SUBAPPLICATION Uebung_039 (* Subapplication Type *)
  (* Standard: 61499-2 *)
  (* Version 1.0, 2023-10-23, franz *)
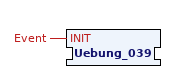
  EVENT_INPUT
    INIT;
  END_EVENT
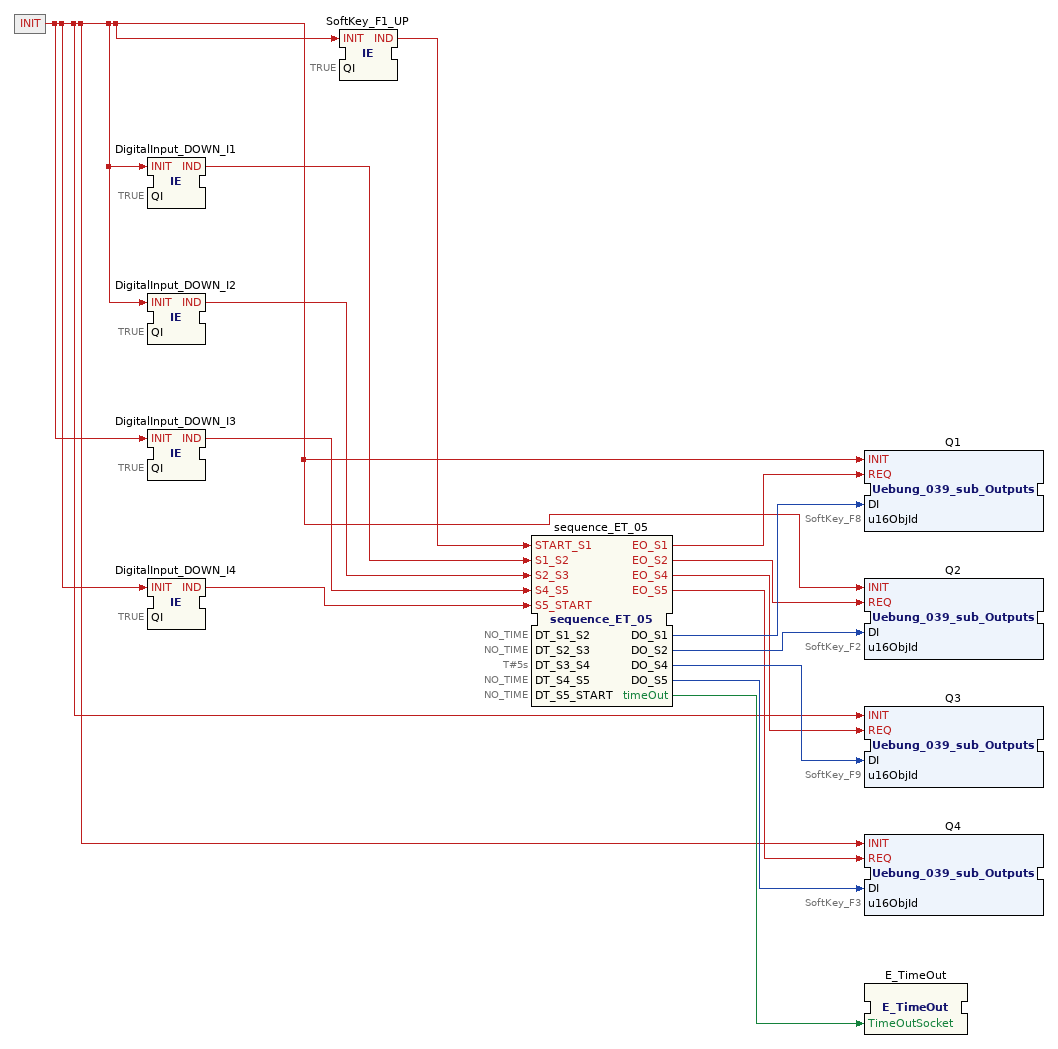
  FBS
    sequence_ET_05 : sequence_ET_05(DT_S1_S2 := NO_TIME, DT_S2_S3 := NO_TIME, DT_S3_S4 := T#5s, DT_S4_S5 := NO_TIME, DT_S5_START := NO_TIME);
    E_TimeOut : E_TimeOut;
    SoftKey_F1_UP : IE(QI := TRUE);
    DigitalInput_DOWN_I1 : IE(QI := TRUE);
    DigitalInput_DOWN_I2 : IE(QI := TRUE);
    DigitalInput_DOWN_I3 : IE(QI := TRUE);
    DigitalInput_DOWN_I4 : IE(QI := TRUE);
  END_FBS
  SUBAPPS
    Q1 : Uebung_039_sub_Outputs(u16ObjId := SoftKey_F8);
    Q2 : Uebung_039_sub_Outputs(u16ObjId := SoftKey_F2);
    Q3 : Uebung_039_sub_Outputs(u16ObjId := SoftKey_F9);
    Q4 : Uebung_039_sub_Outputs(u16ObjId := SoftKey_F3);
  END_SUBAPPS
  EVENT_CONNECTIONS
    INIT TO Q1.INIT;
    INIT TO Q2.INIT;
    INIT TO Q3.INIT;
    INIT TO Q4.INIT;
    sequence_ET_05.EO_S1 TO Q1.REQ;
    sequence_ET_05.EO_S2 TO Q2.REQ;
    sequence_ET_05.EO_S4 TO Q3.REQ;
    sequence_ET_05.EO_S5 TO Q4.REQ;
    INIT TO SoftKey_F1_UP.INIT;
    INIT TO DigitalInput_DOWN_I1.INIT;
    INIT TO DigitalInput_DOWN_I2.INIT;
    INIT TO DigitalInput_DOWN_I3.INIT;
    INIT TO DigitalInput_DOWN_I4.INIT;
    SoftKey_F1_UP.IND TO sequence_ET_05.START_S1;
    DigitalInput_DOWN_I1.IND TO sequence_ET_05.S1_S2;
    DigitalInput_DOWN_I2.IND TO sequence_ET_05.S2_S3;
    DigitalInput_DOWN_I3.IND TO sequence_ET_05.S4_S5;
    DigitalInput_DOWN_I4.IND TO sequence_ET_05.S5_START;
  END_CONNECTIONS
  DATA_CONNECTIONS
    sequence_ET_05.DO_S1 TO Q1.DI;
    sequence_ET_05.DO_S2 TO Q2.DI;
    sequence_ET_05.DO_S4 TO Q3.DI;
    sequence_ET_05.DO_S5 TO Q4.DI;
  END_CONNECTIONS
  ADAPTER_CONNECTIONS
    sequence_ET_05.timeOut TO E_TimeOut.TimeOutSocket;
  END_CONNECTIONS
END_SUBAPPLICATION
